
// ===== library: MasterCopy "maniobra_grabado_secado" =====

FUNCTION_BLOCK "maniobra_grabado_secado"   // FB3, STL
{ S7_Optimized_Access := 'TRUE' }
VERSION : 0.1
BEGIN
END_FUNCTION_BLOCK

// ===== library: MasterCopy "maniobra_cinta" =====

FUNCTION_BLOCK "maniobra_cinta"   // FB5, STL
{ S7_Optimized_Access := 'TRUE' }
VERSION : 0.1
BEGIN
END_FUNCTION_BLOCK

// ===== library: MasterCopy "maniobra_entrada_estacion" =====

FUNCTION_BLOCK "maniobra_entrada_estacion"   // FB7, STL
{ S7_Optimized_Access := 'TRUE' }
VERSION : 0.1
BEGIN
END_FUNCTION_BLOCK